FUNCTION_BLOCK logiBUS_AI_ID (* Input service interface function block for double word input data *)
  (* Description: Copyright (c) 2017 fortiss GmbH, HR Agrartechnik GmbH This program and the accompanying materials are made available under the terms of the Eclipse Public License 2.0 which is available at https://www.eclipse.org/legal/epl-2.0/ SPDX-License-Identifier: EPL-2.0 if AnalogInput_hysteresis = 0, then TimeDelta cannot be 0. set TimeDelta to 16#FFFFFFFF to deactivate cyclic processing, and onyl indicate Changes in Value. *)
  (* Version 1.1, 2026-04-19, Franz Höpfinger, HR Agrartechnik GmbH *)
  (* Version 1.0, 2017-03-20, Monika Wenger, fortiss GmbH *)
  PACKAGE logiBUS::io::AI;
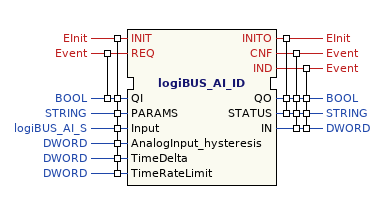
  EVENT_INPUT
    INIT : EInit WITH QI, PARAMS, Input, AnalogInput_hysteresis, TimeDelta, TimeRateLimit; (* Service Initialization *)
    REQ WITH QI; (* Service Request *)
  END_EVENT
  EVENT_OUTPUT
    INITO : EInit WITH QO, STATUS; (* Initialization Confirm *)
    CNF WITH QO, STATUS, IN; (* Confirmation of Requested Service *)
    IND WITH QO, STATUS, IN; (* Indication from Resource *)
  END_EVENT
  VAR_INPUT
    QI : BOOL; (* Event Input Qualifier *)
    PARAMS : STRING; (* Service Parameters *)
    Input : logiBUS::io::AI::logiBUS_AI_S := logiBUS_AI::Invalid; (* Identify the Input Input_I1..I8 *)
    AnalogInput_hysteresis : DWORD;
    TimeDelta : DWORD := 250; (* After How many ms an IND (poll interval) *)
    TimeRateLimit : DWORD := 100; (* Maximum 1 IND in how many ms. (< delta) *)
  END_VAR
  VAR_OUTPUT
    QO : BOOL; (* Event Output Qualifier *)
    STATUS : STRING; (* Service Status *)
    IN : DWORD; (* Input data from resource *)
  END_VAR
END_FUNCTION_BLOCK
